# B&R Automation Studio project EFI (part 27)

#### FunctionsTests.c
```c
/********************************************************************
 * COPYRIGHT -- Bernecker + Rainer
 ********************************************************************
 * Program: ConsentsTests
 * Author: Jorge Murria
 ********************************************************************
 * Prepare machine with basic test to allow proper behabior
 * and starting tasks
 ********************************************************************/

#include <bur/plctypes.h>

#ifdef _DEFAULT_INCLUDES
#include <AsDefault.h>
#endif

#include "UnitTest.h"

#include <stdio.h>
#include <unistd.h>
#include <time.h>         /* clock_t, clock, CLOCKS_PER_SEC */

_LOCAL TIME TimeLast;
_LOCAL TIME endtime;
_LOCAL UDINT diff_t;
_LOCAL STRING stringAux[120];

_LOCAL UINT sensorPosition;

#define FALSE 0
#define TRUE 1

void nextState(){
	exTimesPreFast = gMachine.St.exec.fast;
	exTimesPreSlow = gMachine.St.exec.slow;
	iTestState++;
	TimeLast = clock_ms();
}

void ResetTrackingArrays(){
	for (iIndexArray = 0; iIndexArray < THICK_MAX_UPDATE_VALUES; iIndexArray++)	{
		xTestMediaDetectionValuesL1[iIndexArray] = FALSE;
	}
	for (iIndexArray = 0; iIndexArray < iMAXTRACKINGARRAY; iIndexArray++)	{
		TestMediaTracking[iIndexArray] = FALSE;
		TestBoolMediaTracking[iIndexArray] = FALSE;
	}
	sensorPosition = 0;
}

void ResetTrackingMediaInside(){
	for (iIndexArray = 0; iIndexArray < THICK_MEDIATRACKING_MAX_MEDIA; iIndexArray++)	{
		TestMediaTrackingInside[iIndexArray].HeadPosition = 0;
		TestMediaTrackingInside[iIndexArray].TailPosition = 0;
		TestMediaTrackingInside[iIndexArray].iIndexMediaEnergy = 0;
		TestMediaTrackingInside[iIndexArray].pMediaEnery = 0;
		TestMediaTrackingInside[iIndexArray].Media = MediaConfigReseted;
	}
	for (iIndexArray = 0; iIndexArray < THICKENERGY_MAX_LAMPS; iIndexArray++)	{
		IntensityOutput[iIndexArray] = 0;
	}
	//USINT[0..THICKENERGY_MAX_PROCESS_ITEMS,0..THICKENERGY_MAX_CROSS_ITEMS]
	for (iIndexProcess = 0; iIndexProcess <= THICKENERGY_MAX_PROCESS_ITEMS; iIndexProcess++)	{
		for (iIndexCross = 0; iIndexCross <= THICKENERGY_MAX_CROSS_ITEMS; iIndexCross++)	{
			EnergyData.iPower[iIndexProcess][iIndexCross] = 0;
		}
	}
}

_TEST test_LoadMediaFromFastDataLine(void)
{
	strcpy(txTest, "test_LoadMediaFromFastDataLine");

//TESTS WITH NO GAP

	// 4 Inputs and 5 outputs (v)
	ResetTrackingArrays();
	xTestMediaDetectionValuesL1[0] = TRUE;
	xTestMediaDetectionValuesL1[1] = TRUE;
	xTestMediaDetectionValuesL1[2] = TRUE;
	xTestMediaDetectionValuesL1[3] = TRUE;

	LoadMediaFromFastDataLine(&xTestMediaDetectionValuesL1,4 , INDEXTRACKING_L1, 5, sensorPosition, &TestMediaTracking);
			TEST_ASSERT(TestMediaTracking[sensorPosition + 0]);
			TEST_ASSERT(TestMediaTracking[sensorPosition + 1]);
			TEST_ASSERT(TestMediaTracking[sensorPosition + 2]);
			TEST_ASSERT(TestMediaTracking[sensorPosition + 3]);
			TEST_ASSERT(TestMediaTracking[sensorPosition + 4]); //If variable is TRUE, the test is correct

	LoadMediaFromFastDataBool(&xTestMediaDetectionValuesL1, 4, 5, sensorPosition, &TestBoolMediaTracking);
			TEST_ASSERT(TestBoolMediaTracking[sensorPosition + 0]);
			TEST_ASSERT(TestBoolMediaTracking[sensorPosition + 1]);
			TEST_ASSERT(TestBoolMediaTracking[sensorPosition + 2]);
			TEST_ASSERT(TestBoolMediaTracking[sensorPosition + 3]);
			TEST_ASSERT(TestBoolMediaTracking[sensorPosition + 4]);

	// 4 Inputs and 6 outputs (v)
	ResetTrackingArrays();
	xTestMediaDetectionValuesL1[0] = TRUE;
	xTestMediaDetectionValuesL1[1] = TRUE;
	xTestMediaDetectionValuesL1[2] = TRUE;
	xTestMediaDetectionValuesL1[3] = TRUE;

	LoadMediaFromFastDataLine(&xTestMediaDetectionValuesL1, 4, INDEXTRACKING_L1, 6, 0, &TestMediaTracking);
			TEST_ASSERT(TestMediaTracking[sensorPosition + 0]);
			TEST_ASSERT(TestMediaTracking[sensorPosition + 1]);
			TEST_ASSERT(TestMediaTracking[sensorPosition + 2]);
			TEST_ASSERT(TestMediaTracking[sensorPosition + 3]);
			TEST_ASSERT(TestMediaTracking[sensorPosition + 4]);
			TEST_ASSERT(TestMediaTracking[sensorPosition + 5]); //If variable is TRUE, the test is correct

	LoadMediaFromFastDataBool(&xTestMediaDetectionValuesL1, 4, 6, sensorPosition, &TestBoolMediaTracking);
			TEST_ASSERT(TestBoolMediaTracking[sensorPosition + 0]);
			TEST_ASSERT(TestBoolMediaTracking[sensorPosition + 1]);
			TEST_ASSERT(TestBoolMediaTracking[sensorPosition + 2]);
			TEST_ASSERT(TestBoolMediaTracking[sensorPosition + 3]);
			TEST_ASSERT(TestBoolMediaTracking[sensorPosition + 4]);
			TEST_ASSERT(TestBoolMediaTracking[sensorPosition + 5]);

//TESTS WITH ONLY ONE GAP

	// 4 Inputs and 6 outputs 1 gap
	ResetTrackingArrays();
	xTestMediaDetectionValuesL1[0] = TRUE;
	xTestMediaDetectionValuesL1[1] = FALSE;
	xTestMediaDetectionValuesL1[2] = TRUE;
	xTestMediaDetectionValuesL1[3] = TRUE;

	LoadMediaFromFastDataLine(&xTestMediaDetectionValuesL1, 4, INDEXTRACKING_L1, 6, 0, &TestMediaTracking);
			TEST_ASSERT(TestMediaTracking[sensorPosition + 0]);
			TEST_ASSERT(!TestMediaTracking[sensorPosition + 1]);
			TEST_ASSERT(TestMediaTracking[sensorPosition + 2]);
			TEST_ASSERT(TestMediaTracking[sensorPosition + 3]);
			TEST_ASSERT(TestMediaTracking[sensorPosition + 4]);
			TEST_ASSERT(TestMediaTracking[sensorPosition + 5]); //If variable is TRUE, the test is correct

	LoadMediaFromFastDataBool(&xTestMediaDetectionValuesL1, 4, 6, sensorPosition, &TestBoolMediaTracking);
			TEST_ASSERT(TestBoolMediaTracking[sensorPosition + 0]);
			TEST_ASSERT(!TestBoolMediaTracking[sensorPosition + 1]);
			TEST_ASSERT(TestBoolMediaTracking[sensorPosition + 2]);
			TEST_ASSERT(TestBoolMediaTracking[sensorPosition + 3]);
			TEST_ASSERT(TestBoolMediaTracking[sensorPosition + 4]);
			TEST_ASSERT(TestBoolMediaTracking[sensorPosition + 5]); //If variable is TRUE, the test is correct

	// 3 Inputs and 7 outputs 1 gap
	ResetTrackingArrays();
	xTestMediaDetectionValuesL1[0] = TRUE;
	xTestMediaDetectionValuesL1[1] = FALSE;
	xTestMediaDetectionValuesL1[2] = TRUE;
	LoadMediaFromFastDataLine(&xTestMediaDetectionValuesL1, 3, INDEXTRACKING_L1, 7, sensorPosition, &TestMediaTracking);
			TEST_ASSERT(TestMediaTracking[sensorPosition + 0]);
			TEST_ASSERT(TestMediaTracking[sensorPosition + 1]);
			TEST_ASSERT(!TestMediaTracking[sensorPosition + 2]);
			TEST_ASSERT(!TestMediaTracking[sensorPosition + 3]);
			TEST_ASSERT(TestMediaTracking[sensorPosition + 4]);
			TEST_ASSERT(TestMediaTracking[sensorPosition + 5]);
			TEST_ASSERT(TestMediaTracking[sensorPosition + 6]); //If a 0 appears somewhere, the test is correct

	LoadMediaFromFastDataBool(&xTestMediaDetectionValuesL1, 3, 7, sensorPosition, &TestBoolMediaTracking);
			TEST_ASSERT(TestBoolMediaTracking[sensorPosition + 0]);
			TEST_ASSERT(TestBoolMediaTracking[sensorPosition + 1]);
			TEST_ASSERT(!TestBoolMediaTracking[sensorPosition + 2]);
			TEST_ASSERT(!TestBoolMediaTracking[sensorPosition + 3]);
			TEST_ASSERT(TestBoolMediaTracking[sensorPosition + 4]);
			TEST_ASSERT(TestBoolMediaTracking[sensorPosition + 5]);
			TEST_ASSERT(TestBoolMediaTracking[sensorPosition + 6]); //If a 0 appears somewhere, the test is correct

	// 6 Inputs and 4 outputs 1 gap
	ResetTrackingArrays();
	xTestMediaDetectionValuesL1[0] = TRUE;
	xTestMediaDetectionValuesL1[1] = FALSE;
	xTestMediaDetectionValuesL1[2] = TRUE;
	xTestMediaDetectionValuesL1[3] = TRUE;
	xTestMediaDetectionValuesL1[4] = TRUE;
	xTestMediaDetectionValuesL1[5] = TRUE;

	LoadMediaFromFastDataLine(&xTestMediaDetectionValuesL1, 6, INDEXTRACKING_L1, 4, 0, &TestMediaTracking);
			TEST_ASSERT(!TestMediaTracking[sensorPosition + 0]);
			TEST_ASSERT(!TestMediaTracking[sensorPosition + 1]);
			TEST_ASSERT(TestMediaTracking[sensorPosition + 2]);
			TEST_ASSERT(TestMediaTracking[sensorPosition + 3]);

	LoadMediaFromFastDataBool(&xTestMediaDetectionValuesL1, 6, 4, sensorPosition, &TestBoolMediaTracking);
			TEST_ASSERT(!TestBoolMediaTracking[sensorPosition + 0]);
			TEST_ASSERT(!TestBoolMediaTracking[sensorPosition + 1]);
			TEST_ASSERT(TestBoolMediaTracking[sensorPosition + 2]);
			TEST_ASSERT(TestBoolMediaTracking[sensorPosition + 3]);

	// 7 Inputs and 3 outputs
	ResetTrackingArrays();
	xTestMediaDetectionValuesL1[0] = TRUE;
	xTestMediaDetectionValuesL1[1] = TRUE;
	xTestMediaDetectionValuesL1[2] = TRUE;
	xTestMediaDetectionValuesL1[3] = TRUE;
	xTestMediaDetectionValuesL1[4] = FALSE;
	xTestMediaDetectionValuesL1[5] = TRUE;
	xTestMediaDetectionValuesL1[6] = TRUE;

	LoadMediaFromFastDataLine(&xTestMediaDetectionValuesL1, 7, INDEXTRACKING_L1, 3, sensorPosition, &TestMediaTracking);
			TEST_ASSERT(TestMediaTracking[sensorPosition + 0]);
			TEST_ASSERT(!TestMediaTracking[sensorPosition + 1]);
			TEST_ASSERT(!TestMediaTracking[sensorPosition + 2]); //If a 0 appears somewhere, the test is correct

	LoadMediaFromFastDataBool(&xTestMediaDetectionValuesL1, 7, 3, sensorPosition, &TestBoolMediaTracking);
			TEST_ASSERT(TestBoolMediaTracking[sensorPosition + 0]);
			TEST_ASSERT(!TestBoolMediaTracking[sensorPosition + 1]);
			TEST_ASSERT(!TestBoolMediaTracking[sensorPosition + 2]); //If a 0 appears somewhere, the test is correct

	// 10 Inputs and 2 outputs
	ResetTrackingArrays();
	xTestMediaDetectionValuesL1[0] = TRUE;
	xTestMediaDetectionValuesL1[1] = TRUE;
	xTestMediaDetectionValuesL1[2] = TRUE;
	xTestMediaDetectionValuesL1[3] = TRUE;
	xTestMediaDetectionValuesL1[4] = TRUE;
	xTestMediaDetectionValuesL1[5] = TRUE;
	xTestMediaDetectionValuesL1[6] = TRUE;
	xTestMediaDetectionValuesL1[7] = FALSE;
	xTestMediaDetectionValuesL1[8] = TRUE;
	xTestMediaDetectionValuesL1[9] = TRUE;

	LoadMediaFromFastDataLine(&xTestMediaDetectionValuesL1, 10, INDEXTRACKING_L1, 2, sensorPosition, &TestMediaTracking);
			TEST_ASSERT(TestMediaTracking[sensorPosition + 0]);
			TEST_ASSERT(!TestMediaTracking[sensorPosition + 1]); //If a 0 appears somewhere, the test is correct

	LoadMediaFromFastDataBool(&xTestMediaDetectionValuesL1, 10, 2, sensorPosition, &TestBoolMediaTracking);
			TEST_ASSERT(TestBoolMediaTracking[sensorPosition + 0]);
			TEST_ASSERT(!TestBoolMediaTracking[sensorPosition + 1]); //If a 0 appears somewhere, the test is correct

	// 2 Inputs and 10 outputs
	ResetTrackingArrays();
	xTestMediaDetectionValuesL1[0] = TRUE;
	xTestMediaDetectionValuesL1[1] = FALSE;

	LoadMediaFromFastDataLine(&xTestMediaDetectionValuesL1, 2, INDEXTRACKING_L1, 10, sensorPosition, &TestMediaTracking);
			TEST_ASSERT(TestMediaTracking[sensorPosition + 0]);
			TEST_ASSERT(TestMediaTracking[sensorPosition + 1]);
			TEST_ASSERT(TestMediaTracking[sensorPosition + 2]);
			TEST_ASSERT(TestMediaTracking[sensorPosition + 3]);
			TEST_ASSERT(!TestMediaTracking[sensorPosition + 4]);
			TEST_ASSERT(!TestMediaTracking[sensorPosition + 5]);
			TEST_ASSERT(!TestMediaTracking[sensorPosition + 6]);
			TEST_ASSERT(!TestMediaTracking[sensorPosition + 7]);
			TEST_ASSERT(!TestMediaTracking[sensorPosition + 8]);
			TEST_ASSERT(!TestMediaTracking[sensorPosition + 9] ); //If a 0 appears somewhere, the test is correct

	LoadMediaFromFastDataBool(&xTestMediaDetectionValuesL1, 2, 10, sensorPosition, &TestBoolMediaTracking);
			TEST_ASSERT(TestBoolMediaTracking[sensorPosition + 0]);
			TEST_ASSERT(TestBoolMediaTracking[sensorPosition + 1]);
			TEST_ASSERT(TestBoolMediaTracking[sensorPosition + 2]);
			TEST_ASSERT(TestBoolMediaTracking[sensorPosition + 3]);
			TEST_ASSERT(!TestBoolMediaTracking[sensorPosition + 4]);
			TEST_ASSERT(!TestBoolMediaTracking[sensorPosition + 5]);
			TEST_ASSERT(!TestBoolMediaTracking[sensorPosition + 6]);
			TEST_ASSERT(!TestBoolMediaTracking[sensorPosition + 7]);
			TEST_ASSERT(!TestBoolMediaTracking[sensorPosition + 8]);
			TEST_ASSERT(!TestBoolMediaTracking[sensorPosition + 9] ); //If a 0 appears somewhere, the test is correct

	// 2 Inputs and 1 outputs
	ResetTrackingArrays();
	xTestMediaDetectionValuesL1[0] = TRUE;
	xTestMediaDetectionValuesL1[1] = FALSE;

	LoadMediaFromFastDataLine(&xTestMediaDetectionValuesL1, 2, INDEXTRACKING_L1, 1, sensorPosition, &TestMediaTracking);
	TEST_ASSERT(!TestMediaTracking[sensorPosition + 0] ); //If a 0 appears somewhere, the test is correct
	LoadMediaFromFastDataBool(&xTestMediaDetectionValuesL1, 2, 1, sensorPosition, &TestBoolMediaTracking);
	TEST_ASSERT(!TestBoolMediaTracking[sensorPosition + 0] ); //If a 0 appears somewhere, the test is correct

	// 5 inputs to 9 outputs
	ResetTrackingArrays();
	xTestMediaDetectionValuesL1[0] = TRUE;
	xTestMediaDetectionValuesL1[1] = FALSE;
	xTestMediaDetectionValuesL1[2] = TRUE;
	xTestMediaDetectionValuesL1[3] = TRUE;
	xTestMediaDetectionValuesL1[4] = TRUE;

	LoadMediaFromFastDataLine(&xTestMediaDetectionValuesL1, 5, INDEXTRACKING_L1, 9, sensorPosition, &TestMediaTracking);
			TEST_ASSERT(TestMediaTracking[sensorPosition + 0]);
			TEST_ASSERT(!TestMediaTracking[sensorPosition + 1]);
			TEST_ASSERT(!TestMediaTracking[sensorPosition + 2]);
			TEST_ASSERT(TestMediaTracking[sensorPosition + 3]);
			TEST_ASSERT(TestMediaTracking[sensorPosition + 4]);
			TEST_ASSERT(TestMediaTracking[sensorPosition + 5]);
			TEST_ASSERT(TestMediaTracking[sensorPosition + 6]);
			TEST_ASSERT(TestMediaTracking[sensorPosition + 7]);
			TEST_ASSERT(TestMediaTracking[sensorPosition + 8] ); //If a 0 appears somewhere, the test is correct

	LoadMediaFromFastDataBool(&xTestMediaDetectionValuesL1, 5, 9, sensorPosition, &TestBoolMediaTracking);
			TEST_ASSERT(TestBoolMediaTracking[sensorPosition + 0]);
			TEST_ASSERT(!TestBoolMediaTracking[sensorPosition + 1]);
			TEST_ASSERT(!TestBoolMediaTracking[sensorPosition + 2]);
			TEST_ASSERT(TestBoolMediaTracking[sensorPosition + 3]);
			TEST_ASSERT(TestBoolMediaTracking[sensorPosition + 4]);
			TEST_ASSERT(TestBoolMediaTracking[sensorPosition + 5]);
			TEST_ASSERT(TestBoolMediaTracking[sensorPosition + 6]);
			TEST_ASSERT(TestBoolMediaTracking[sensorPosition + 7]);
			TEST_ASSERT(TestBoolMediaTracking[sensorPosition + 8] ); //If a 0 appears somewhere, the test is correct

	//9 inputs to 5 outputs
	ResetTrackingArrays();
	xTestMediaDetectionValuesL1[0] = TRUE;
	xTestMediaDetectionValuesL1[1] = TRUE;
	xTestMediaDetectionValuesL1[2] = TRUE;
	xTestMediaDetectionValuesL1[3] = TRUE;
	xTestMediaDetectionValuesL1[4] = FALSE;
	xTestMediaDetectionValuesL1[5] = TRUE;
	xTestMediaDetectionValuesL1[6] = TRUE;
	xTestMediaDetectionValuesL1[7] = TRUE;
	xTestMediaDetectionValuesL1[8] = TRUE;

	LoadMediaFromFastDataLine(&xTestMediaDetectionValuesL1, 9, INDEXTRACKING_L1, 5, sensorPosition, &TestMediaTracking);
			TEST_ASSERT(TestMediaTracking[sensorPosition + 0]);
			TEST_ASSERT(TestMediaTracking[sensorPosition + 1]);
			TEST_ASSERT(!TestMediaTracking[sensorPosition + 2]);
			TEST_ASSERT(TestMediaTracking[sensorPosition + 3]);
			TEST_ASSERT(TestMediaTracking[sensorPosition + 4]); //If a 0 appears somewhere, the test is correct

	LoadMediaFromFastDataBool(&xTestMediaDetectionValuesL1, 9, 5, sensorPosition, &TestBoolMediaTracking);
			TEST_ASSERT(TestBoolMediaTracking[sensorPosition + 0]);
			TEST_ASSERT(TestBoolMediaTracking[sensorPosition + 1]);
			TEST_ASSERT(!TestBoolMediaTracking[sensorPosition + 2]);
			TEST_ASSERT(TestBoolMediaTracking[sensorPosition + 3]);
			TEST_ASSERT(TestBoolMediaTracking[sensorPosition + 4]); //If a 0 appears somewhere, the test is correct

	//7 inputs to 6 outputs
	ResetTrackingArrays();
	xTestMediaDetectionValuesL1[0] = TRUE;
	xTestMediaDetectionValuesL1[1] = TRUE;
	xTestMediaDetectionValuesL1[2] = TRUE;
	xTestMediaDetectionValuesL1[3] = TRUE;
	xTestMediaDetectionValuesL1[4] = FALSE;
	xTestMediaDetectionValuesL1[5] = TRUE;
	xTestMediaDetectionValuesL1[6] = TRUE;

	LoadMediaFromFastDataLine(&xTestMediaDetectionValuesL1, 7, INDEXTRACKING_L1, 6, sensorPosition, &TestMediaTracking);
			TEST_ASSERT(TestMediaTracking[sensorPosition + 0]);
			TEST_ASSERT(TestMediaTracking[sensorPosition + 1]);
			TEST_ASSERT(TestMediaTracking[sensorPosition + 2]);
			TEST_ASSERT(!TestMediaTracking[sensorPosition + 3]);
			TEST_ASSERT(!TestMediaTracking[sensorPosition + 4]);
			TEST_ASSERT(TestMediaTracking[sensorPosition + 5]); //If variable is TRUE, the test is correct

	LoadMediaFromFastDataBool(&xTestMediaDetectionValuesL1, 7, 6, sensorPosition, &TestBoolMediaTracking);
			TEST_ASSERT(TestBoolMediaTracking[sensorPosition + 0]);
			TEST_ASSERT(TestBoolMediaTracking[sensorPosition + 1]);
			TEST_ASSERT(TestBoolMediaTracking[sensorPosition + 2]);
			TEST_ASSERT(!TestBoolMediaTracking[sensorPosition + 3]);
			TEST_ASSERT(!TestBoolMediaTracking[sensorPosition + 4]);
			TEST_ASSERT(TestBoolMediaTracking[sensorPosition + 5]); //If variable is TRUE, the test is correct

	//6 inputs to 7 outputs
	ResetTrackingArrays();
	xTestMediaDetectionValuesL1[0] = TRUE;
	xTestMediaDetectionValuesL1[1] = TRUE;
	xTestMediaDetectionValuesL1[2] = FALSE;
	xTestMediaDetectionValuesL1[3] = TRUE;
	xTestMediaDetectionValuesL1[4] = TRUE;
	xTestMediaDetectionValuesL1[5] = TRUE;

	LoadMediaFromFastDataLine(&xTestMediaDetectionValuesL1, 6, INDEXTRACKING_L1, 7, sensorPosition, &TestMediaTracking);
			TEST_ASSERT(TestMediaTracking[sensorPosition + 0]);
			TEST_ASSERT(TestMediaTracking[sensorPosition + 1]);
			TEST_ASSERT(!TestMediaTracking[sensorPosition + 2]);
			TEST_ASSERT(TestMediaTracking[sensorPosition + 3]);
			TEST_ASSERT(TestMediaTracking[sensorPosition + 4]);
			TEST_ASSERT(TestMediaTracking[sensorPosition + 5]);
			TEST_ASSERT(TestMediaTracking[sensorPosition + 6]); //If variable is TRUE, the test is correct

	LoadMediaFromFastDataBool(&xTestMediaDetectionValuesL1, 6, 7, sensorPosition, &TestBoolMediaTracking);
			TEST_ASSERT(TestBoolMediaTracking[sensorPosition + 0]);
			TEST_ASSERT(TestBoolMediaTracking[sensorPosition + 1]);
			TEST_ASSERT(!TestBoolMediaTracking[sensorPosition + 2]);
			TEST_ASSERT(TestBoolMediaTracking[sensorPosition + 3]);
			TEST_ASSERT(TestBoolMediaTracking[sensorPosition + 4]);
			TEST_ASSERT(TestBoolMediaTracking[sensorPosition + 5]);
			TEST_ASSERT(TestBoolMediaTracking[sensorPosition + 6]); //If variable is TRUE, the test is correct

	//10 to 1 (limit case)
	ResetTrackingArrays();
	xTestMediaDetectionValuesL1[0] = TRUE;
	xTestMediaDetectionValuesL1[1] = TRUE;
	xTestMediaDetectionValuesL1[2] = TRUE;
	xTestMediaDetectionValuesL1[3] = TRUE;
	xTestMediaDetectionValuesL1[4] = FALSE;
	xTestMediaDetectionValuesL1[5] = TRUE;
	xTestMediaDetectionValuesL1[6] = TRUE;
	xTestMediaDetectionValuesL1[7] = TRUE;
	xTestMediaDetectionValuesL1[8] = TRUE;
	xTestMediaDetectionValuesL1[9] = TRUE;

	LoadMediaFromFastDataLine(&xTestMediaDetectionValuesL1, 10, INDEXTRACKING_L1, 1, sensorPosition, &TestMediaTracking);
			TEST_ASSERT(!TestMediaTracking[sensorPosition + 0]);//a 0 must appear
	LoadMediaFromFastDataBool(&xTestMediaDetectionValuesL1, 10, 1, sensorPosition, &TestBoolMediaTracking);
			TEST_ASSERT(!TestBoolMediaTracking[sensorPosition + 0]);//a 0 must appear

	//10 to 3 with one gap
	ResetTrackingArrays();
	xTestMediaDetectionValuesL1[0] = TRUE;
	xTestMediaDetectionValuesL1[1] = TRUE;
	xTestMediaDetectionValuesL1[2] = TRUE;
	xTestMediaDetectionValuesL1[3] = TRUE;
	xTestMediaDetectionValuesL1[4] = TRUE;
	xTestMediaDetectionValuesL1[5] = TRUE;
	xTestMediaDetectionValuesL1[6] = TRUE;
	xTestMediaDetectionValuesL1[7] = FALSE;
	xTestMediaDetectionValuesL1[8] = TRUE;
	xTestMediaDetectionValuesL1[9] = TRUE;

	LoadMediaFromFastDataLine(&xTestMediaDetectionValuesL1, 10, INDEXTRACKING_L1, 3, sensorPosition, &TestMediaTracking);
			TEST_ASSERT(TestMediaTracking[sensorPosition + 0]);
			TEST_ASSERT(TestMediaTracking[sensorPosition + 1]);
			TEST_ASSERT(!TestMediaTracking[sensorPosition + 2]);//a 0 must appear

	LoadMediaFromFastDataBool(&xTestMediaDetectionValuesL1, 10, 3, sensorPosition, &TestBoolMediaTracking);
			TEST_ASSERT(TestBoolMediaTracking[sensorPosition + 0]);
			TEST_ASSERT(TestBoolMediaTracking[sensorPosition + 1]);
			TEST_ASSERT(!TestBoolMediaTracking[sensorPosition + 2]);//a 0 must appear

	//This 2 lines just for the last TestCase
	strcpy(txTest, "test_TestCase Finished!! Congrats!");
	strcpy(txStateDesc, "--");
	TEST_DONE;
}

_TEST test_RevMediaTrackingEnergyInPos(void)
{
	strcpy(txTest, "test_RevMediaTrackingEnergyInPos");

	//Dry just in one side. Image displaced
	ResetTrackingMediaInside();
	TestMediaTrackingInside[0].HeadPosition = 2;
	TestMediaTrackingInside[0].TailPosition = 0;
	TestMediaTrackingInside[0].pMediaEnery = &EnergyData;

	EnergyData.iPower[0][0] = 100;

	RevMediaTrackingEnergyInPos(&TestMediaTrackingInside, 1,
		1, 2,
		48, 1400.0/48.0, -1400.0/2, 0,
		0, IntensityOutput);
	TEST_ASSERT(IntensityOutput[24] == 100);

	//Dry just in one side. Image centered
	ResetTrackingMediaInside();
	TestMediaTrackingInside[0].HeadPosition = 2;
	TestMediaTrackingInside[0].TailPosition = 0;
	TestMediaTrackingInside[0].pMediaEnery = &EnergyData;
	TestMediaTrackingInside[0].Media.rLength = 100;
	TestMediaTrackingInside[0].Media.rWidth = 1400;
	TestMediaTrackingInside[0].Media.rCrossOffset = -700;
	TestMediaTrackingInside[0].Media.rDocLength = 100;
	TestMediaTrackingInside[0].Media.rDocWidth = 1400;
	TestMediaTrackingInside[0].Media.rDocCrossOffset = -700;

	EnergyData.iPower[0][0] = 100;

	RevMediaTrackingEnergyInPos(&TestMediaTrackingInside, 1,
		1, 2,
		48, 1400.0/48.0, -1400.0/2, 0,
		0, IntensityOutput);
	TEST_ASSERT(IntensityOutput[48] == 100);

	//Dry just in one side. Image centered
	ResetTrackingMediaInside();
	TestMediaTrackingInside[0].HeadPosition = 2;
	TestMediaTrackingInside[0].TailPosition = 0;
	TestMediaTrackingInside[0].pMediaEnery = &EnergyData;
	TestMediaTrackingInside[0].Media.rLength = 100;
	TestMediaTrackingInside[0].Media.rWidth = 1400;
	TestMediaTrackingInside[0].Media.rCrossOffset = -700;
	TestMediaTrackingInside[0].Media.rDocLength = 100;
	TestMediaTrackingInside[0].Media.rDocWidth = 1400;
	TestMediaTrackingInside[0].Media.rDocCrossOffset = -700;

	EnergyData.iPower[0][139] = 100;

	RevMediaTrackingEnergyInPos(&TestMediaTrackingInside, 1,
		1, 2,
		48, 1400.0/48.0, -1400.0/2, 0,
		0, IntensityOutput);
	TEST_ASSERT(IntensityOutput[1] == 100);

	//Dry in the center. Image centered. Without overlap
	ResetTrackingMediaInside();
	TestMediaTrackingInside[0].HeadPosition = 2;
	TestMediaTrackingInside[0].TailPosition = 0;
	TestMediaTrackingInside[0].pMediaEnery = &EnergyData;
	TestMediaTrackingInside[0].Media.rLength = 100;
	TestMediaTrackingInside[0].Media.rWidth = 1400;
	TestMediaTrackingInside[0].Media.rCrossOffset = -700;
	TestMediaTrackingInside[0].Media.rDocLength = 100;
	TestMediaTrackingInside[0].Media.rDocWidth = 1400;
	TestMediaTrackingInside[0].Media.rDocCrossOffset = -700;

	EnergyData.iPower[0][69] = 100;
	EnergyData.iPower[0][70] = 100;
	EnergyData.iPower[0][71] = 100;

	RevMediaTrackingEnergyInPos(&TestMediaTrackingInside, 1,
		1, 2,
		48, 1400.0/48.0, -1400.0/2, 0,
		0, IntensityOutput);
	TEST_ASSERT(IntensityOutput[23] == 0);
	TEST_ASSERT(IntensityOutput[24] == 100);
	TEST_ASSERT(IntensityOutput[25] == 100);
	TEST_ASSERT(IntensityOutput[26] == 0);

	//Dry in the center. Image centered. WITH overlap
	ResetTrackingMediaInside();
	TestMediaTrackingInside[0].HeadPosition = 2;
	TestMediaTrackingInside[0].TailPosition = 0;
	TestMediaTrackingInside[0].pMediaEnery = &EnergyData;
	TestMediaTrackingInside[0].Media.rLength = 100;
	TestMediaTrackingInside[0].Media.rWidth = 1400;
	TestMediaTrackingInside[0].Media.rCrossOffset = -700;
	TestMediaTrackingInside[0].Media.rDocLength = 100;
	TestMediaTrackingInside[0].Media.rDocWidth = 1400;
	TestMediaTrackingInside[0].Media.rDocCrossOffset = -700;

	EnergyData.iPower[0][69] = 100;
	EnergyData.iPower[0][70] = 100;
	EnergyData.iPower[0][71] = 100;

	RevMediaTrackingEnergyInPos(&TestMediaTrackingInside, 1,
		1, 2,
		48, 1400.0/48.0, -1400.0/2, 10,
		0, IntensityOutput);
	TEST_ASSERT(IntensityOutput[22] == 0);
	TEST_ASSERT(IntensityOutput[23] == 100);
	TEST_ASSERT(IntensityOutput[24] == 100);
	TEST_ASSERT(IntensityOutput[25] == 100);
	TEST_ASSERT(IntensityOutput[26] == 0);

	//Dry in the center. Image centered. Without overlap. SAW
	ResetTrackingMediaInside();
	TestMediaTrackingInside[0].HeadPosition = 2;
	TestMediaTrackingInside[0].TailPosition = 0;
	TestMediaTrackingInside[0].pMediaEnery = &EnergyData;
	TestMediaTrackingInside[0].Media.rLength = 100;
	TestMediaTrackingInside[0].Media.rWidth = 1400;
	TestMediaTrackingInside[0].Media.rCrossOffset = -700;
	TestMediaTrackingInside[0].Media.rDocLength = 100;
	TestMediaTrackingInside[0].Media.rDocWidth = 1400;
	TestMediaTrackingInside[0].Media.rDocCrossOffset = -700;

	EnergyData.iPower[0][57] = 40;
	EnergyData.iPower[0][58] = 45;
	EnergyData.iPower[0][59] = 50;
	EnergyData.iPower[0][60] = 55;
	EnergyData.iPower[0][61] = 60;
	EnergyData.iPower[0][62] = 65;
	EnergyData.iPower[0][63] = 70;
	EnergyData.iPower[0][64] = 75;
	EnergyData.iPower[0][65] = 80;
	EnergyData.iPower[0][66] = 85;
	EnergyData.iPower[0][67] = 90;
	EnergyData.iPower[0][68] = 95;
	EnergyData.iPower[0][69] = 100;
	EnergyData.iPower[0][70] = 100;
	EnergyData.iPower[0][71] = 95;
	EnergyData.iPower[0][72] = 90;
	EnergyData.iPower[0][73] = 85;
	EnergyData.iPower[0][74] = 80;
	EnergyData.iPower[0][75] = 75;
	EnergyData.iPower[0][76] = 70;
	EnergyData.iPower[0][77] = 65;
	EnergyData.iPower[0][78] = 60;
	EnergyData.iPower[0][79] = 55;
	EnergyData.iPower[0][80] = 50;
	EnergyData.iPower[0][81] = 45;
	EnergyData.iPower[0][82] = 40;

	RevMediaTrackingEnergyInPos(&TestMediaTrackingInside, 1,
		1, 2,
		48, 1400.0/48.0, -1400.0/2, 0,
		0, IntensityOutput);
	TEST_ASSERT(IntensityOutput[19] == 0);
	TEST_ASSERT(IntensityOutput[20] == 45);
	TEST_ASSERT(IntensityOutput[21] == 60);
	TEST_ASSERT(IntensityOutput[22] == 75);
	TEST_ASSERT(IntensityOutput[23] == 90);
	TEST_ASSERT(IntensityOutput[24] == 100);
	TEST_ASSERT(IntensityOutput[25] == 100);
	TEST_ASSERT(IntensityOutput[26] == 90);
	TEST_ASSERT(IntensityOutput[27] == 75);
	TEST_ASSERT(IntensityOutput[28] == 60);
	TEST_ASSERT(IntensityOutput[29] == 45);
	TEST_ASSERT(IntensityOutput[30] == 0);

	//Dry in the center. Image centered. WITH overlap. SAW
	ResetTrackingMediaInside();
	TestMediaTrackingInside[0].HeadPosition = 2;
	TestMediaTrackingInside[0].TailPosition = 0;
	TestMediaTrackingInside[0].pMediaEnery = &EnergyData;
	TestMediaTrackingInside[0].Media.rLength = 100;
	TestMediaTrackingInside[0].Media.rWidth = 1400;
	TestMediaTrackingInside[0].Media.rCrossOffset = -700;
	TestMediaTrackingInside[0].Media.rDocLength = 100;
	TestMediaTrackingInside[0].Media.rDocWidth = 1400;
	TestMediaTrackingInside[0].Media.rDocCrossOffset = -700;

	EnergyData.iPower[0][57] = 40;
	EnergyData.iPower[0][58] = 45;
	EnergyData.iPower[0][59] = 50;
	EnergyData.iPower[0][60] = 55;
	EnergyData.iPower[0][61] = 60;
	EnergyData.iPower[0][62] = 65;
	EnergyData.iPower[0][63] = 70;
	EnergyData.iPower[0][64] = 75;
	EnergyData.iPower[0][65] = 80;
	EnergyData.iPower[0][66] = 85;
	EnergyData.iPower[0][67] = 90;
	EnergyData.iPower[0][68] = 95;
	EnergyData.iPower[0][69] = 100;
	EnergyData.iPower[0][70] = 100;
	EnergyData.iPower[0][71] = 95;
	EnergyData.iPower[0][72] = 90;
	EnergyData.iPower[0][73] = 85;
	EnergyData.iPower[0][74] = 80;
	EnergyData.iPower[0][75] = 75;
	EnergyData.iPower[0][76] = 70;
	EnergyData.iPower[0][77] = 65;
	EnergyData.iPower[0][78] = 60;
	EnergyData.iPower[0][79] = 55;
	EnergyData.iPower[0][80] = 50;
	EnergyData.iPower[0][81] = 45;
	EnergyData.iPower[0][82] = 40;

	RevMediaTrackingEnergyInPos(&TestMediaTrackingInside, 1,
		1, 2,
		48, 1400.0/48.0, -1400.0/2, 10,
		0, IntensityOutput);
	TEST_ASSERT(IntensityOutput[19] == 0);
	TEST_ASSERT(IntensityOutput[20] == 50);
	TEST_ASSERT(IntensityOutput[21] == 65);
	TEST_ASSERT(IntensityOutput[22] == 80);
	TEST_ASSERT(IntensityOutput[23] == 95);
	TEST_ASSERT(IntensityOutput[24] == 100);
	TEST_ASSERT(IntensityOutput[25] == 100);
	TEST_ASSERT(IntensityOutput[26] == 95);
	TEST_ASSERT(IntensityOutput[27] == 80);
	TEST_ASSERT(IntensityOutput[28] == 65);
	TEST_ASSERT(IntensityOutput[29] == 50);
	TEST_ASSERT(IntensityOutput[30] == 0);

	//Dry just minimum
	ResetTrackingMediaInside();
	TestMediaTrackingInside[0].HeadPosition = 2;
	TestMediaTrackingInside[0].TailPosition = 0;
	TestMediaTrackingInside[0].pMediaEnery = &EnergyData;
	TestMediaTrackingInside[0].Media.rLength = 100;
	TestMediaTrackingInside[0].Media.rWidth = 1400;
	TestMediaTrackingInside[0].Media.rCrossOffset = -700;
	TestMediaTrackingInside[0].Media.rDocLength = 100;
	TestMediaTrackingInside[0].Media.rDocWidth = 1400;
	TestMediaTrackingInside[0].Media.rDocCrossOffset = -700;

	EnergyData.iPower[0][0] = 0;

	RevMediaTrackingEnergyInPos(&TestMediaTrackingInside, 1,
		1, 2,
		48, 1400.0/48.0, -1400.0/2, 0,
		15, IntensityOutput);
	TEST_ASSERT(IntensityOutput[1] == 15);
	TEST_ASSERT(IntensityOutput[48] == 15);

	//Dry just in one side. Image centered. Image delayed
	ResetTrackingMediaInside();
	TestMediaTrackingInside[0].HeadPosition = 10;
	TestMediaTrackingInside[0].TailPosition = 0;
	TestMediaTrackingInside[0].pMediaEnery = &EnergyData;
	TestMediaTrackingInside[0].Media.rLength = 1500;
	TestMediaTrackingInside[0].Media.rWidth = 1400;
	TestMediaTrackingInside[0].Media.rCrossOffset = -700;
	TestMediaTrackingInside[0].Media.rDocLength = 1500;
	TestMediaTrackingInside[0].Media.rDocWidth = 1400;
	TestMediaTrackingInside[0].Media.rDocCrossOffset = -700;

	// 29 = 29position * 5cm = 145cm (cofigured 150cm)
	EnergyData.iPower[29][0] = 100;

	RevMediaTrackingEnergyInPos(&TestMediaTrackingInside, 1,
		-150, 1,
		48, 1400.0/48.0, -1400.0/2, 0,
		0, &IntensityOutput);
	TEST_ASSERT(IntensityOutput[48] == 100);

	TEST_DONE;
}

_TEST test_ShiftArrayForwardOffset(void)
{
	strcpy(txTest, "test_ShiftArrayForwardOffset");

	// Assign data
	for (iIndexArray = 0; iIndexArray < iMAXTRACKINGARRAY; iIndexArray++)	{
		TestMediaTracking[iIndexArray] = iIndexArray;
	}

	TestMediaTracking[0] = TestMediaTracking[1000]; //Copying the value of a large index to later comparing
	ShiftArrayOffset(&TestMediaTracking, sizeof(TestMediaTracking), sizeof(TestMediaTracking[0]), 1, 3, iMAXTRACKINGARRAY-3);

	TEST_ASSERT_EQUAL_INT(TestMediaTracking[1], TestMediaTracking[3]);
	TEST_ASSERT_EQUAL_INT(TestMediaTracking[1000 + 3 - 1], TestMediaTracking[0]);

	ResetTrackingMediaInside();
	MediaData = MediaConfigReseted;
	MediaData.id = 1;
	MediaData.iLine = 1;
	MediaData.rCrossOffset = -700;
	MediaData.rDocCrossOffset = -600;
	MediaData.rDocLength = 1500;
	MediaData.rDocProcessOffset = 0;
	MediaData.rDocWidth = 1200;
	MediaData.rLength = 1500;
	MediaData.rThickness = 2;
	MediaData.rWidth = 1400;

	Stack_iTotalNewMedia = 0;
	EnergyRack_iIndex = 1;

	udResult = AssignLastItemEnergyInStack(
		&MediaData,
		&EnergyData,
		&NewMediaStack,
		&MediaEnergyRack,
		&Stack_iTotalNewMedia,
		&EnergyRack_iIndex
		);

	TEST_ASSERT_EQUAL_INT(0 , udResult);
	TEST_ASSERT_EQUAL_INT(1 , Stack_iTotalNewMedia);

	MediaData = MediaConfigReseted;
	MediaData.id = 2;
	MediaData.iLine = 1;
	MediaData.rCrossOffset = -700;
	MediaData.rDocCrossOffset = -600;
	MediaData.rDocLength = 1500;
	MediaData.rDocProcessOffset = 0;
	MediaData.rDocWidth = 1200;
	MediaData.rLength = 1500;
	MediaData.rThickness = 2;
	MediaData.rWidth = 1400;

	udResult = AssignLastItemEnergyInStack(
		&MediaData,
		&EnergyData,
		&NewMediaStack,
		&MediaEnergyRack,
		&Stack_iTotalNewMedia,
		&EnergyRack_iIndex
		);

	TEST_ASSERT_EQUAL_INT(0 , udResult);
	TEST_ASSERT_EQUAL_INT(2 , Stack_iTotalNewMedia);

	// Error trying to insert a media with the same Id
	udResult = CheckNotItemInStack(
		MediaData.id,
		&NewMediaStack,
		Stack_iTotalNewMedia,
		&Stack_iTotalNewMediaPos);
	TEST_ASSERT_EQUAL_INT(1520 , udResult); //Extected an error because the Id.2 is already in the list

	// Function to insert
	MediaData = MediaConfigReseted;
	MediaData.id = 3;
	MediaData.iLine = 1;
	MediaData.rCrossOffset = -700;
	MediaData.rDocCrossOffset = -600;
	MediaData.rDocLength = 1500;
	MediaData.rDocProcessOffset = 0;
	MediaData.rDocWidth = 1200;
	MediaData.rLength = 1500;
	MediaData.rThickness = 2;
	MediaData.rWidth = 1400;

	// Check the position of the Id=1
	udResult = CheckItemInStack(
		1,
		&NewMediaStack,
		&Stack_iTotalNewMedia,
		&Stack_iTotalNewMediaPos
		);
	TEST_ASSERT_EQUAL_INT(0, udResult); // Everything went OK
	TEST_ASSERT_EQUAL_INT(0, Stack_iTotalNewMediaPos); // Everything went OK

	udResult = InsertItemEnergyInStack(
		1,
		&MediaData,
		&EnergyData,
		&NewMediaStack,
		&MediaEnergyRack,
		&Stack_iTotalNewMedia,
		&EnergyRack_iIndex
		);
	TEST_ASSERT_EQUAL_INT(0, udResult); // Everything went OK
	TEST_ASSERT_EQUAL_INT(3, NewMediaStack[1].Media.id); // The Third media is in the second position

	// Function to remove
	udResult = RemoveItemInStack(
		1,
		&NewMediaStack,
		&Stack_iTotalNewMedia);
	TEST_ASSERT_EQUAL_INT(0, udResult); // Everything went OK
	TEST_ASSERT_EQUAL_INT(2, NewMediaStack[1].Media.id); // The second media is in the second position again

	udResult = RemoveItemInStack(
		-1,
		&NewMediaStack,
		&Stack_iTotalNewMedia);
	TEST_ASSERT_EQUAL_INT(0, udResult); // Everything went OK
	TEST_ASSERT_EQUAL_INT(0, Stack_iTotalNewMedia); // The list is emptyed
	TEST_ASSERT_EQUAL_INT(0, NewMediaStack[0].Media.id); // The list is emptyed

	// Assign data
	for (iIndexArray = 0; iIndexArray < iMAXTRACKINGARRAY; iIndexArray++)	{
		TestMediaTracking[iIndexArray] = 0;
	}

	//This 2 lines just for the last TestCase
	strcpy(txTest, "test_FunctionTests Finished!! Congrats!");
	strcpy(txStateDesc, "--");
	TEST_DONE;
}

/*
B+R UnitTest: This is generated code.
Do not edit! Do not move!
Description: UnitTest Testprogramm infrastructure (TestSet).
LastUpdated: 2024-03-07 09:14:50Z
By B+R UnitTest Helper Version: 2.0.1.59
*/
UNITTEST_FIXTURES(fixtures)
{
	new_TestFixture("test_LoadMediaFromFastDataLine", test_LoadMediaFromFastDataLine),
	new_TestFixture("test_RevMediaTrackingEnergyInPos", test_RevMediaTrackingEnergyInPos),
	new_TestFixture("test_ShiftArrayForwardOffset", test_ShiftArrayForwardOffset),
};

UNITTEST_CALLER_COMPLETE_EXPLICIT(FunctionsTests, "FunctionsTests", 0, 0, fixtures, 0, 0, 0);
```

### Tests.var
```iecst
VAR
	iTestState : USINT;
	testPassedAsserts : UDINT;
	xSometestFailedAsserts : BOOL;
	testFailedAsserts : UDINT;
	txTest : STRING[80];
	txStateDesc : STRING[80];
	exTimesPreFast : UDINT;
	exTimesPreSlow : UDINT;
	diffExecFast : UDINT;
	iIndexBlock : USINT;
	iIndex : USINT;
	iIndexPrepareCuring : USINT;
	iInksChillerIndex : USINT;
	iIndexPsuOk : USINT;
	iCheckInkStartedIndex : USINT;
	rPreviousVacPressureSp : REAL;
	rPreviousBlockMotorPosition : REAL;
END_VAR
```

### Program Logical/UnitTest/Tests/TemplateTests (ANSIC)

#### autoGeneratedFile.c - Auto generated code
```c
/*
B+R UnitTest: This is generated code.
Do not edit! Do not move!
Description: UnitTest Testprogramm infrastructure (List of TestSets).
LastUpdated: 2020-05-18 14:29:28Z
By B+R UnitTest Helper Version: 2.0.1.59
*/
#include "UnitTest.h"

UNITTEST_TESTSET_DECLARATION  TemplateTests;

UNITTEST_TESTSET_FIXTURES(utTestSets)
{
	new_TestSet(TemplateTests),
};
UNTITTEST_TESTSET_HANDLER();
```

- ReplicateTest.bat (not shown)

- Visualisation Logical/mappView (not shown)

- JsonCheck.bat (not shown)

- Doc Editor. Marktext.url (not shown)

- UaExpertConnections.uap (not shown)

- B&R System Diagnostics Manager Dryer.url (not shown)

- mapp View diagnostic Dryer.url (not shown)

- mapp View diagnostic Printer.url (not shown)

Listed in the project but not available here: Logical/Libraries/BRSE_JSON/BRSE_JSON.fun, Logical/Libraries/BRSE_JSON/BRSE_JSON.c, Logical/Libraries/BRSE_JSON/BRSE_JSON_Main.h, Logical/Libraries/BRSE_JSON/version_history.c, Logical/Libraries/ErrACS380/Types.typ, Logical/Libraries/ErrACS380/ErrACS380.fun, Logical/ExtPack/_Ancillaries/FeederCtrl/FeederCtrl_v1/FeederCtrl/Feeder.st, Logical/ExtPack/_Ancillaries/FeederCtrl/FeederCtrl_v1/FeederCtrl/Status.st, Logical/ExtPack/_Ancillaries/FeederCtrl/FeederCtrl_v1/FeederCtrl/Configuration.st, Logical/ExtPack/_Ancillaries/FeederCtrl/FeederCtrl_v1/FeederCtrl/Alarms.st, Logical/ExtPack/_Ancillaries/FeederCtrl/FeederCtrl_v1/Feeder.typ, Logical/ExtPack/_Ancillaries/PrimerCtrl/PrimerCtrl_v1/PrimerCtrl/Status.st, Logical/ExtPack/_Ancillaries/PrimerCtrl/PrimerCtrl_v1/PrimerCtrl/Alarms.st, Logical/ExtPack/_Ancillaries/PrimerCtrl/PrimerCtrl_v1/PrimerCtrl/AssignDataComms.st, Logical/ExtPack/_Ancillaries/PrimerCtrl/PrimerSim/PrimerSim_v1/PrimerSim, Logical/ExtPack/_Ancillaries/PrimerCtrl/PrimerSim/PrimerSim_v1/PrimerSim.typ, Logical/ExtPack/_Ancillaries/StackerCtrl/StackerSim/StackerSim_v1/StackerSim/StackerSim.var, Logical/ExtPack/_Ancillaries/StackerCtrl/StackerSim/StackerSim_v1/StackerSim.typ, Logical/ExtPack/_Comms/ModbusComms/ModbusComms_v1/Libraries/BRSE_MBT/BRSE_MBT.var, Logical/ExtPack/_Comms/ModbusComms/ModbusComms_v1/Libraries/BRSE_MBT/BRSE_MBT.fun, Logical/ExtPack/_Comms/ModbusComms/ModbusComms_v1/Libraries/BRSE_MBT/Version_History.c, Logical/ExtPack/_Comms/ModbusComms/ModbusComms_v1/Libraries/BRSE_MBT/BRSE_MBT_Main.h, Logical/ExtPack/_Comms/ModbusComms/ModbusComms_v1/Libraries/BRSE_MBT/MBT_Client.c, Logical/ExtPack/_Comms/ModbusComms/ModbusComms_v1/Libraries/BRSE_MBT/Example_Server.c, Logical/ExtPack/_Cure/ArcLampGEW/ArcLampGew_v1/ArcLampGewCtrl/ArcLampGew.st, Logical/ExtPack/_Cure/ArcLampGEW/ArcLampGew_v1/ArcLampGewCtrl/State.st, Logical/ExtPack/_Cure/ArcLampGEW/ArcLampGew_v1/ArcLampGewCtrl/Comms.st, Logical/ExtPack/_Cure/ArcLampGEW/ArcLampGew_v1/ArcLampGewCtrl/AlarmsSummary.st, Logical/ExtPack/_Cure/ArcLampGEW/ArcLampGew_v1/ArcLampGewCtrl/Calculations.st, Logical/ExtPack/_Cure/ArcLampGEW/ArcLampGew_v1/ArcLampGewCtrl/Outputs.st, Logical/ExtPack/_Cure/ArcLampGEW/ArcLampGew_v1/ArcLampGewCtrl/EventLog.st, Logical/ExtPack/_Cure/ArcLampGEW/ArcLampSim/ArcLampSim_v1/ArcLampSim/ArcLampSim.st, Logical/ExtPack/_Cure/ArcLampGEW/ArcLampSim/ArcLampSim_v1/ArcLampSim/Comms.st, Logical/ExtPack/_Cure/CuringLedCtrl/CuringLedSim/CuringLedSim_v1/CuringLedSim/CuringLedSim.var, Logical/ExtPack/_Cure/CuringLedCtrl/CuringLedSim/CuringLedSim_v1/InitCuringLedSim/InitCuringLedSim.st, Logical/ExtPack/_Cure/NIRAdphos/NIRAdphos_v1/NIRAdphosCtrl/NIRAdphosCtrl.st, Logical/ExtPack/_Cure/NIRAdphos/NIRAdphos_v1/NIRAdphosCtrl/Calculations.st, Logical/ExtPack/_Cure/NIRAdphos/NIRAdphos_v1/NIRAdphosCtrl/Alarms.st, Logical/ExtPack/_Cure/NIRAdphos/NIRAdphos_v1/NIRAdphosCtrl/AlarmsSummary.st, Logical/ExtPack/_Cure/NIRAdphos/NIRAdphos_v1/NIRAdphosCtrl/CommsNir1.var, Logical/ExtPack/_Cure/NIRAdphos/NIRAdphos_v1/NIRAdphosCtrl/CommsNir2.var, Logical/ExtPack/_Cure/NIRAdphos/NIRAdphos_v1/NIRAdphosCtrl/LocalFunctions.fun, Logical/ExtPack/_Cure/NIRAdphos/NIRAdphos_v1/NIRAdphosCtrl/NirFunctions.st, Logical/ExtPack/_Cure/NIRAdphos/NIRAdphos_v1/NIRAdphosCtrl/CommsBase.st, Logical/ExtPack/_Cure/NIRAdphos/NIRAdphos_v1/NIRAdphosCtrl.typ, Logical/ExtPack/_Cure/NIRAdphos/NIRAdphos_v1/Documentation, Logical/ExtPack/_Cure/NIRAdphos/NirAdphosSim/NirAdphosSim_v1/NirAdphosSim.typ, Logical/ExtPack/_Extras/ChillerCtrl/ChillerCtrl_v2/ChillerCtrl/Chiller.st, Logical/ExtPack/_Extras/ChillerCtrl/ChillerCtrl_v2/ChillerCtrl/ChillerCtrl.st, Logical/ExtPack/_Extras/ChillerCtrl/ChillerCtrl_v2/InitChiller/InitChiller.st, Logical/ExtPack/_Extras/ChillerCtrl/ChillerSim/ChillerSim_v1/ChillerSim, Logical/ExtPack/_Extras/ChillerCtrl/ChillerSim/ChillerSim_v1/InitChillerSim, Logical/ExtPack/_Extras/PowerMeterCtrl/PowerMeterCtrl_v1/InitPowerMeterCtrl/InitPowerMeterCtrl.st, Logical/ExtPack/_Extras/PowerMeterCtrl/PowerMeterCtrl_v1/PowerMeter.var, Logical/ExtPack/_Extras/PowerMeterCtrl/PowerMeterCtrl_v1/PowerMeterCtrl.typ, Logical/ExtPack/_Extras/SafetyControllerCtrl/SafetyControllerCtrl_v1/SafetyControllerCtrl/SafetyController.st, Logical/ExtPack/_Extras/SafetyControllerCtrl/SafetyControllerSim/SafetyControllerSim_v1/SafetyControllerSim/SafetyControllerSim.st, Logical/ExtPack/_Media/ThicknessCtrl/ThicknessCtrl_v2/ThicknessCtrl_Fast, Logical/ExtPack/_Media/ThicknessCtrl/ThicknessCtrl_v2/ThicknessCtrl.typ, Logical/ExtPack/_Media/nSensorCtrl/nSensorCtrl_v2/nSensorCtrl/Motors.st, Logical/ExtPack/_Media/nSensorCtrl/nSensorCtrl_v2/nSensorCtrl/MachineState.st, Logical/ExtPack/_Media/nSensorCtrl/nSensorCtrl_v2/nSensorCtrl/EventLog.st, Logical/ExtPack/_Media/nSensorCtrl/nSensorCtrl_v2/nSensorCtrl/nSensorCtrl.var, Logical/ExtPack/_Media/nSensorCtrl/nSensorCtrl_v2/nSensorCtrl_Fast, Logical/ExtPack/_Media/nSensorCtrl/nSensorCtrl_v2/nSensorCtrl.typ, Logical/ExtPack/_Media/AnalogThicknessCtrl/AnalogThicknessCtrl_v1/AnalogThickness/AnalogThickness.st, Logical/ExtPack/_Media/AnalogThicknessCtrl/AnalogThicknessCtrl_v1/AnalogThickness/EventLog.st, Logical/ExtPack/_Media/AnalogThicknessCtrl/AnalogThicknessCtrl_v1/AnalogThickness/Alarms.st, Logical/ExtPack/_Media/AnalogThicknessCtrl/AnalogThicknessCtrl_v1/AnalogThickness/AlarmSounds.st, Logical/ExtPack/_Motion/AxisCtrl/AxisCtrl_v2/AxisCtrl/InitSequence.st, Logical/ExtPack/_Motion/AxisCtrl/AxisCtrl_v2/AxisCtrl/StateSupervisor.st, Logical/ExtPack/_Motion/AxisCtrl/AxisCtrl_v2/AxisCtrl/AxisCtrl.var, Logical/ExtPack/_Motion/AxisCtrl/AxisCtrl_v2/InitAxisControl/InitAxisControl.st, Logical/ExtPack/_Motion/IclaCtrl/IclaCtrl_v4/IclaCtrl/Icla.st, Logical/ExtPack/_Motion/IclaCtrl/IclaCtrl_v4/IclaCtrl/IclaSDO.st, Logical/ExtPack/_Motion/IclaCtrl/IclaCtrl_v4/IclaCtrl/Variables.var, Logical/ExtPack/_Motion/IclaCtrl/IclaSim/IclaSim_v1/IclaSim, Logical/ExtPack/_Motion/IclaCtrl/IclaSim/IclaSim_v1/IclaSim.typ, Logical/ExtPack/_Motion/IclaCtrl/IclaSim/IclaSim_v1/IclaSimGen.var, Logical/ExtPack/_Motion/InverterCtrl/InverterCtrl_v1/InverterCtrl/Simulation.st, Logical/ExtPack/_Motion/InverterCtrl/InverterCtrl_v1/InverterCtrl/ErrorTable.st, Logical/ExtPack/_Motion/InverterCtrl/InverterCtrl_v1/InverterCtrl/ResetComms.st, Logical/ExtPack/_Motion/InverterCtrl/InverterCtrl_v1/Inverter.typ, Logical/ExtPack/_Tools/EventLog/EventLog_v1/EventLogGen/EventLog.st, Logical/ExtPack/_Tools/EventLog/EventLog_v1/EventLogGen/EventLog.fun, Logical/ExtPack/_Tools/EventLog/EventLog_v1/EvLogLib/EvLogLib.fun, Logical/ExtPack/_Tools/EventLog/EventLog_v1/EvLogLib/EvLog.typ, Logical/ExtPack/_Tools/EventLog/EventLog_v1/EvLogLib/EventLoader.st, Logical/ExtPack/_Tools/TestBench/TraySim/TraySim_v1/TraySim/Main.st, Logical/ExtPack/_Tools/TestBench/TraySim/TraySim_v1/InitTraySim, Logical/ExtPack/_Tools/TestBench/TraySim/TraySim_v1/TraySimGen.var, Logical/ExtPack/_Transport/BeltCleaning/BeltCleaning_v1/BeltCleaning/GeneralLogic.st, Logical/ExtPack/_Transport/BeltCleaning/BeltCleaning_v1/BeltCleaning/Alarms.st, Logical/ExtPack/_Transport/BeltCleaning/BeltCleaning_v1/BeltCleaning/Outputs.st, Logical/ExtPack/_Transport/BeltCleaning/BeltCleaning_v1/BeltCleaning/BeltClean.var, Logical/ExtPack/_Transport/BeltCleaning/BeltCleaningSim/BeltCleaningSim/BeltCleanSim.var, Logical/ExtPack/_Transport/BeltCtrl/BeltCtrl_v1/BeltCtrl/Alarms.st, Logical/ExtPack/_Transport/BeltCtrl/BeltCtrl_v1/BeltCtrl/ResetAlarms.st, Logical/ExtPack/_Transport/BeltCtrl/BeltCtrl_v1/BeltCtrl/EventLog.st, Logical/ExtPack/_Transport/BeltCtrl/BeltCtrl_v1/BeltCtrl/BeltManager.var, Logical/ExtPack/_Transport/EdgeHoldDown/EdgeHoldDown_v1/EdgeHoldDown.typ, Logical/ExtPack/_Transport/JamDetectCtrl/JamDetect_v1/JamDetect.typ, Logical/ExtPack/_Transport/JamDetectCtrl/JamDetect_v1/JamDetect.var, Logical/ExtPack/_Transport/PairedIclaMotors/PairedIclaMotorsSim/PairedIclaMotorsSim_v1/PairedIclaMotorsSim/PairedIclaMotorsSim.st, Logical/ExtPack/_Transport/PairedIclaMotors/PairedIclaMotorsSim/PairedIclaMotorsSim_v1/PairedIclaMotorsSim/PairedIclaMotorsSim.var, Logical/ExtPack/_Transport/PairedIclaMotors/PairedIclaMotorsSim/PairedIclaMotorsSim_v1/InitPairedIclaMotorsSim.var, Logical/ExtPack/_Transport/TransVacuumCtrl/TransVacuumCtrl_v1/InitTransVacuumCtrl, Logical/ExtPack/_Transport/TransVacuumCtrl/TransVacuumCtrl_v1/TransVacuum.typ, Logical/ExtPack/_Transport/TransVacuumCtrl/TransVacuumCtrl_v1/TransVacuum.var, Logical/ExtPack/_Transport/TransVacuumCtrl/TransVacuumSim/TransVacuumSim_v1/TransVacuumSim/Main.st, Logical/ExtPack/BlockCtrl/BlockCtrl_v1/BlockCtrl/BlockManager.st, Logical/ExtPack/BlockCtrl/BlockCtrl_v1/BlockCtrl/Inputs.st, Logical/ExtPack/BlockCtrl/BlockCtrl_v1/BlockCtrl/BlockAlarms.st, Logical/ExtPack/BlockCtrl/BlockCtrl_v1/BlockCtrl/InksGetSet.st, Logical/ExtPack/BlockCtrl/BlockCtrl_v1/BlockCtrl/BlockStateGen.st, Logical/ExtPack/BlockCtrl/BlockCtrl_v1/BlockCtrl/ManualLogic.st, Logical/ExtPack/BlockCtrl/BlockCtrl_v1/BlockCtrl/InputParamsMotors.st, Logical/ExtPack/BlockCtrl/BlockCtrl_v1/BlockCtrl/ValvesUnit.st, Logical/ExtPack/BlockCtrl/BlockCtrl_v1/BlockCtrl/EventLog.st, Logical/ExtPack/BlockCtrl/BlockCtrl_v1/BlockCtrl/BlockCtrl.var, Logical/ExtPack/BlockCtrl/BlockCtrl_v1/InitBlockCtrl/InitiBlock.st, Logical/ExtPack/BlockCtrl/BlockCtrl_v1/Block.typ, Logical/ExtPack/BlockCtrl/BlockCtrl_v1/Block.var, Logical/ExtPack/InksCtrl/InksCtrl_v3/InitInksCtrl/Types.typ, Logical/ExtPack/InksCtrl/InksCtrl_v3/InitInksCtrl/Variables.var, Logical/ExtPack/InksCtrl/InksCtrl_v3/InksCtrl/Main.st, Logical/ExtPack/InksCtrl/InksCtrl_v3/InksCtrl/inkLevel.st, Logical/ExtPack/InksCtrl/InksCtrl_v3/InksCtrl/controlMode.st, Logical/ExtPack/InksCtrl/InksCtrl_v3/InksCtrl/calculations.st, Logical/ExtPack/InksCtrl/InksCtrl_v3/InksCtrl/dripControl.st, Logical/ExtPack/InksCtrl/InksCtrl_v3/InksCtrl/startUp.st, Logical/ExtPack/InksCtrl/InksCtrl_v3/InksCtrl/reservoirMode.st, Logical/ExtPack/InksCtrl/InksCtrl_v3/InksCtrl/tempControl.st, Logical/ExtPack/InksCtrl/InksCtrl_v3/InksCtrl/solenoids.st, Logical/ExtPack/InksCtrl/InksCtrl_v3/InksCtrl/powPrintHeads.st, Logical/ExtPack/InksCtrl/InksCtrl_v3/InksCtrl/alarmsSummary.st, Logical/ExtPack/InksCtrl/InksCtrl_v3/InksCtrl/alarmsSound.st, Logical/ExtPack/InksCtrl/InksCtrl_v3/InksCtrl/pressPosAcceleration.st, Logical/ExtPack/InksCtrl/InksCtrl_v3/InksCtrl/Inks.fun, Logical/ExtPack/InksCtrl/InksCtrl_v3/InksCtrl/PIDParams.st, Logical/ExtPack/InksCtrl/InksCtrl_v3/InksCtrl/InksCtrl.var, Logical/ExtPack/InksCtrl/InksCtrl_v3/InksCtrl/Constants.var, Logical/ExtPack/InksCtrl/InksSim/InksSim_v1/InitInksSim/InitInks.st, Logical/ExtPack/SimpleBlockCtrl/SimpleBlockCtrl_v1/SimpleBlockCtrl/BlockManager.st, Logical/ExtPack/SimpleBlockCtrl/SimpleBlockCtrl_v1/SimpleBlockCtrl/BlockParameters.st, Logical/ExtPack/SimpleBlockCtrl/SimpleBlockCtrl_v1/SimpleBlockCtrl/AlarmSound.st, Logical/ExtPack/SimpleBlockCtrl/SimpleBlockCtrl_v1/SimpleBlockCtrl/AlarmsSummary.st, Logical/ExtPack/SimpleBlockCtrl/SimpleBlockCtrl_v1/SimpleBlockCtrl/ResetAlarms.st, Logical/ExtPack/SimpleBlockCtrl/SimpleBlockCtrl_v1/SimpleBlockCtrl/ControlState.st, Logical/ExtPack/SimpleBlockCtrl/SimpleBlockCtrl_v1/SimpleBlockCtrl/BlockStatesCtrl.st, Logical/ExtPack/SimpleBlockCtrl/SimpleBlockCtrl_v1/SimpleBlockCtrl/BlockStateMach.st, Logical/ExtPack/SimpleBlockCtrl/SimpleBlockCtrl_v1/SimpleBlockCtrl/BlockStateGen.st, Logical/ExtPack/SimpleBlockCtrl/SimpleBlockCtrl_v1/SimpleBlockCtrl/GeneralLogic.st, Logical/ExtPack/SimpleBlockCtrl/SimpleBlockCtrl_v1/SimpleBlockCtrl/AutoLogic.st, Logical/ExtPack/SimpleBlockCtrl/SimpleBlockCtrl_v1/SimpleBlockCtrl/EventLog.st, Logical/ExtPack/SimpleBlockCtrl/SimpleBlockCtrl_v1/SimpleBlockCtrl/LogicFunctions.st, Logical/ExtPack/SimpleBlockCtrl/SimpleBlockCtrl_v1/SimpleBlockCtrl.typ, Logical/ExtPack/SimpleBlockCtrl/SimpleBlockCtrl_v1/SimpleBlockCtrl.var, Logical/ExtPack/SimpleBlockCtrl/SimpleBlockSim/SimpleBlockSim_v1/SimpleBlockSim/BlockSim.var, Logical/GStructs/Dryer.typ, Logical/GStructs/InksBox.typ, Logical/GVars/Global_IO.var, Logical/GVars/Global.var, Logical/GVars/MotionBasis.var, Logical/GVars/GlobalComms.var, Logical/GVars/Simulation.var, Logical/Printer/Comms/PLC2Kernel, Logical/Printer/Comms/Kernel2PLC, Logical/Printer/Comms/Comms.var, Logical/Printer/Config/MachineConfigurator/MachineModel.st, Logical/Printer/Config/MachineConfigurator/AsignCommonData.st, Logical/Printer/Config/MachineConfigurator/AsignDataP4.st, Logical/Printer/Config/MachineConfigurator/AsignDataP5.st, Logical/Printer/Config/MachineConfigurator/AsignDataShld.st, Logical/Printer/Config/MachineConfigurator/AsignDataCube.st, Logical/Printer/Config/MachineConfigurator/AssignDataMecano.st, Logical/Printer/Config/MachineConfigurator/AsignDataPlcDiagnosis.st, Logical/Printer/Config/MachineConfigurator/JamSensorsAssignation.st, Logical/Printer/InksSignals/InksInputs/printHeadBaseData.st, Logical/Printer/InksSignals/InksInputs/printHeadNozomi2.st, Logical/Printer/InksSignals/InksInputs/printHeadNozomi2Mineral.st, Logical/Printer/Sim/SimMachine/Initialization.st, Logical/Printer/Sim/SimMachine/MachineModelCode.st, Logical/Printer/Sim/SimMachine/General.st, Logical/Printer/Sim/SimMachine/UPS.st, Logical/Printer/Sim/SimMachine/Tests.st, Logical/Printer/Sim/SimMachine/TestEventLog.st, Logical/Printer/Sim/SimMachine_Fast/Media.st, Logical/Printer/Sim/SimMachine_Fast/Stack.st, Logical/Printer/Sim/SimMachine_Fast/SimMachine_Fast.var, Logical/Printer/Sim/SimMachine.typ, Logical/Printer/Sim/SimMachineGen.var, Logical/Printer/Sim/TestResources/TestResources.var, Logical/Dryer/DryerComms.var, Logical/Dryer/DryerRemote.typ, Logical/Dryer/Config/Initialize/Initialize.st, Logical/Dryer/Config/MachineConfigurator/MachineConfigurator.st, Logical/Dryer/Config/MachineConfigurator/AsignCommonData.st, Logical/Dryer/Config/MachineConfigurator/AsignDataDryerNoz2.st, Logical/Dryer/Config/SavePermanent/SavePermanent.st, Logical/Dryer/DryerCtrl/DryerCtrl_Fast/DryerCtrl_Fast.st, Logical/Dryer/DryerCtrl/DryerCtrl_Fast/DryerState.st, Logical/Dryer/DryerCtrl/DryerCtrl_Fast/AutoLocal.st, Logical/Dryer/DryerCtrl/DryerCtrl_Fast/OrdersDryer.st, Logical/Dryer/DryerCtrl/DryerCtrl_Fast/Alarms.st, Logical/Dryer/DryerCtrl/DryerCtrl_Fast/AlarmsSummary.st, Logical/Dryer/DryerCtrl/DryerCtrl_Fast/EventLog.st, Logical/Dryer/DryerCtrl/DryerCtrl_Fast/DryerCtrl_Fast.var, Logical/Dryer/DryerCtrl/DryerCtrl_Slow/GeneralMachineData.st, Logical/Dryer/DryerCtrl/DryerCtrl_Slow/CleanBelt.st, Logical/Dryer/DryerCtrl/DryerCtrl_Slow/AlarmsSlow.st, Logical/Dryer/DryerCtrl/DryerCtrl_Slow/SoundBeacon.st, Logical/Dryer/DryerCtrl/DryerCtrl_Slow/Constants.var, Logical/Dryer/PhysicalMapping/PhysicalMapInputs/MappingInputs.st, Logical/Dryer/PhysicalMapping/PhysicalMapOutputs/OutputsDryerNoz2.st, Logical/Dryer/Documentation/Sensors, Logical/Dryer/DryerSimAnc/DryerSimAnc_v1/DryerSimAnc/DryerSimAnc.st, Logical/Dryer/DryerSimAnc/DryerSimAnc_v1/DryerSimAnc/DryerSimAnc.var, Logical/AxisTables/BeltS1400_a, Logical/AxisTables/BeltS1400_i, Logical/AxisTables/BeltP5_a, Logical/AxisTables/BeltShield_a, Logical/AxisTables/BeltShield_i, Logical/AxisTables/BK1_i, Logical/AxisTables/NonCrash_i, Logical/AxisTables/BeltNozomi2_i, Logical/AxisTables/BK1_Nozomi2_a, Logical/AxisTables/BK1_Nozomi2_i, Logical/AxisTables/Belt17000_i, Logical/AxisTables/BK_17000_i, Logical/InkBox/Config/Initialize, Logical/InkBox/Config/SavePermanent/SavePermanent.st, Logical/InkBox/HMI/HMI/Alarms.st, Logical/InkBox/PhysicalMapping/PhysicalMapInputs/MappingInputs.st, Logical/InkBox/Transport/Transport/Transport.st, Logical/InkBox/Transport/Transport/Transport.var, Logical/UnitTest/Dryer/PrepareDryer/testSuite.c, Logical/UnitTest/Dryer/BeltTests/BeltTests.c, Logical/UnitTest/Dryer/BeltTests/BeltTests.var, Logical/UnitTest/Dryer/BeltTests/testSuite.c, Logical/UnitTest/Libraries/UnitTest/UnitTest.h, Logical/UnitTest/Libraries/LibAssert1/LibAssert1.h, Logical/UnitTest/Libraries/LibAssert1/LibAssert1_ThresholdAssert.h, Logical/UnitTest/Libraries/LibAssert1/LibAssert1_ThresholdAssert.c, Logical/UnitTest/Libraries/LibAssert1/LibAssert1_REAL_ArrayAsserts.h, Logical/UnitTest/Tests/PrePrepare/PrePrepare.c, Logical/UnitTest/Tests/PrePrepare/PrePrepare.var, Logical/UnitTest/Tests/PrePrepare/testSuite.c, Logical/UnitTest/Tests/PrepareMachine/autoGeneratedFile.c, Logical/UnitTest/Tests/BlockTests/BlockTests.c, Logical/UnitTest/Tests/BlockTests/testSuite.c, Logical/UnitTest/Tests/BlockTests/BlockTests.var, Logical/UnitTest/Tests/BlockTests/autoGeneratedFile.c, Logical/UnitTest/Tests/CleaningTests/CleaningTests.var, Logical/UnitTest/Tests/CleaningTests/testSuite.c, Logical/UnitTest/Tests/CleaningTests/autoGeneratedFile.c, Logical/UnitTest/Tests/TrVacuumTests/testSuite.c, Logical/UnitTest/Tests/LineTests/LineTests.c, Logical/UnitTest/Tests/LineTests/LineTests.var, Logical/UnitTest/Tests/LineTests/testSuite.c, Logical/UnitTest/Tests/LineTests/autoGeneratedFile.c, Logical/UnitTest/Tests/TemplateTests/TemplateTests.c, Logical/UnitTest/Tests/TemplateTests/TemplateTests.var, Logical/UnitTest/Tests/TemplateTests/testSuite.c
